// TIA Portal V19 export
TYPE "PPrf_Generic"
// stored: Access Published
   STRUCT
      Material_Width : Real;   // [mm] Larghezza materiale del rotolo
      Material_Thickness : Real;   // [mm] Spessore materiale = Spessore finale del pezzo
      Material_Tol_Min : Real;   // [mm] Tolleranza minima materiale (usato da sensore di controllo)
      Material_Tol_Max : Real;   // [mm] Tolleranza massima materiale (usato da sensore di controllo)
      Beam_Code : Int;   // Codice Pezzo: 0= SG formato da una singola parte; 1= C/S = Formato da due parti accoppiate
      Beam_W_A_Code : Int;   // Codice Larghezza Pezzo = Altezza impilamento. Esempio 40 = 40mm; 45 = 45 mm. (HMI symbolic IO Field)
      Beam_H_B_Code : Int;   // Codice Altezza Pezzo = Base impilamento. Esempio 60 = 60mm; 120 = 120mm. (HMI symbolic IO Field)
      Beam_TK_Code : Int;   // Codice Spessore. Valori possibili 125 = 1,25 mm; 150 = 1,5 mm; 200 = 2,00 mm (HMI symbolic IO Field)
      Beam_Len_Tol_Min : Real;   // [mm] Tolleranza minima lunghezza pezzi
      Beam_Len_Tol_Max : Real;   // [mm] Tolleranza massima lunghezza pezzi
      Thickness_Mark : Int;   // 0-1 esecuzione del marchio di identificazione spessore
      Trace_Mark : Int;   // 0-1 esecuzione del marchio di tracciabilità (numero colata rotolo usato)
      Option_1 : Int;   // Free option 1
      Option_2 : Int;   // Free option 2
      PackLayout_BeamsPerLayer : Int;   // Schema di impilamento = Quantità pezzi per strato
      PackLayout_Layers_Qty : Int;   // Schema di impilamento = Quantità strati
   END_STRUCT;
END_TYPE
